INTERFACE I_NodeLinks EXTENDS I_Disposable

METHOD PUBLIC Clear
VAR_INPUT
END_VAR
END_METHOD

METHOD PUBLIC Create : I_NodeLink
VAR_INPUT
	LinkId : T_MAXSTRING;
	LinkSourceNode : I_Node;
	LinkSource : I_LinkSource;
	LinkDestinationNode : I_Node;
	LinkDestination : I_LinkDestination;
END_VAR
END_METHOD

METHOD PUBLIC DisconnectAll
VAR_INPUT
END_VAR
END_METHOD

METHOD PUBLIC GetKeyValueEnumerator : I_KeyValueForwardEnumerator
VAR_INPUT
END_VAR
END_METHOD

METHOD PUBLIC TryGetLinkById : BOOL
VAR_INPUT
	Id : T_MAXSTRING;
	Destination : REFERENCE TO I_NodeLink;
END_VAR
END_METHOD

END_INTERFACE

(* stored: Version 1.1.0.1, ProductVersion 3.1.4024.13
   Itf I_NodeLinks: Id {6342794e-42d2-001e-2efc-85604cd854b5}
   Method Clear: Id {30be076b-3530-0564-1530-c4e83f34bf2c}
   Method Create: Id {5fe0ede6-ad42-0634-1240-887245e47764}
   Method DisconnectAll: Id {8bba65c9-be92-0e81-37df-f0a1695700db}
   Method GetKeyValueEnumerator: Id {926d330e-86bb-06ab-2c14-0e61d4530fdc}
   Method TryGetLinkById: Id {4fb5c24f-9a54-0758-1aab-a8aa5d7c222a} *)
